Fanuc KAREL source: kd00056.KL

-- PROVISIONAL review KL for V770-1; original PC SHA256 6f99078cd79b9f985d637f846ba1e0369a6bd70511608936fb09b2118e443344
-- Incomplete behavior may be omitted. Consult companion uncertainty JSON. Do not deploy.
PROGRAM KD00056
%NOLOCKGROUP
VAR
  I : INTEGER
  J : INTEGER
  B : BOOLEAN
  R : REAL
  S : STRING[80]
-- UNRESOLVED_DECL P type=000101
BEGIN
  -- UNRESOLVED_PC offsets 5-37; opcodes 01,22,1C,06,82,03,9D,9C,9D,12,9D,1B,9D,13,04,0B
  -- UNRESOLVED_PC offsets 42-46; opcodes 7F
END KD00056
